Fanuc KAREL source: kt00072.KL

-- PROVISIONAL review KL for V1013-1; original PC SHA256 e2c3dde6fd39597e60a879110ccd32f4bf2f9381f6891360c5c18db4b639e178
-- Incomplete behavior may be omitted. Consult companion uncertainty JSON. Do not deploy.
PROGRAM KT00072
%NOLOCKGROUP
VAR
  I1 : INTEGER
  OUT : REAL
-- UNRESOLVED_DECL H2 type=002017
BEGIN
  -- UNRESOLVED_PC offsets 5-16; opcodes 2E,23
  -- UNRESOLVED_PC offsets 21-35; opcodes 2E,22,9D,33,B4
  -- UNRESOLVED_PC offsets 40-63; opcodes 21,22,9D,33,B3,54,64,23
  -- UNRESOLVED_PC offsets 68-72; opcodes 7F
END KT00072
